// Mitsubishi GX Works2 project: guide_kommunikasjon_master   PLC: Q00

// global labels: Global1
VAR_GLOBAL
  tank AT D0 : INT;
  slider AT D20 : INT;
  knapp_0 AT M20 : BOOL;
  knapp_1 AT M21 : BOOL;
  lampe_0 AT M100 : BOOL;
  lampe_1 AT M101 : BOOL;
  avFlagg_0 AT M0 : BOOL;
  avFlagg_1 AT M1 : BOOL;
  paFlagg_0 AT M10 : BOOL;
  paFlagg_1 AT M11 : BOOL;
END_VAR

// task Task_01 (event TRUE, interval 0, priority 31): POU_01

PROGRAM POU_01
(* structured ladder/FBD written out as ST: instructions are called as NAME(EN, inputs, outputs); _pN, _eN, _tN stand for wires *)
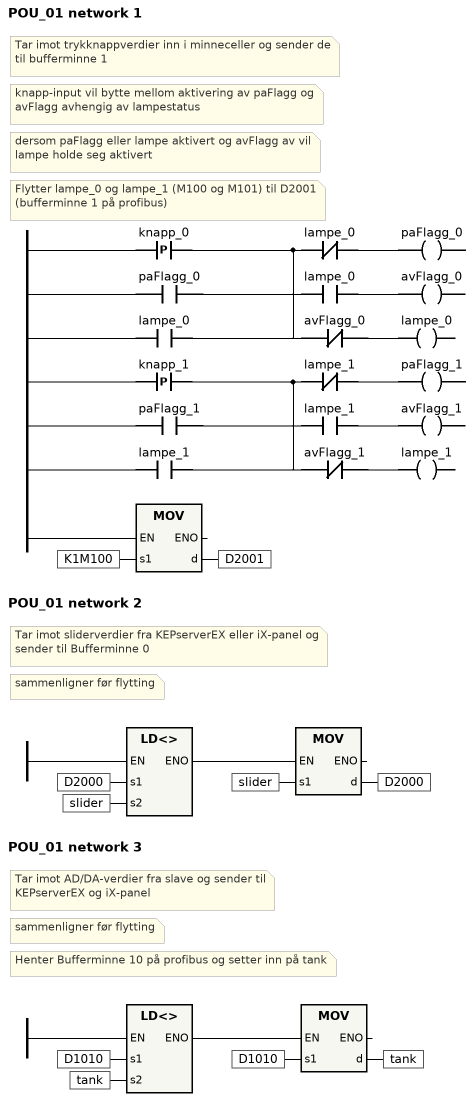
(* network 1 *)
(* Tar imot trykknappverdier inn i minneceller og sender de til bufferminne 1 *)
(* knapp-input vil bytte mellom aktivering av paFlagg og avFlagg avhengig av lampestatus *)
(* dersom paFlagg eller lampe aktivert og avFlagg av vil lampe holde seg aktivert *)
(* Flytter lampe_0 og lampe_1 (M100 og M101) til D2001 (bufferminne 1 på profibus) *)
_p1 := LDP(TRUE, knapp_0);
paFlagg_0 := _p1 AND NOT lampe_0;
avFlagg_0 := _p1 AND lampe_0;
lampe_0 := (paFlagg_0 OR lampe_0) AND NOT avFlagg_0;
_p2 := LDP(TRUE, knapp_1);
paFlagg_1 := _p2 AND NOT lampe_1;
avFlagg_1 := _p2 AND lampe_1;
lampe_1 := (paFlagg_1 OR lampe_1) AND NOT avFlagg_1;
MOV(TRUE, K1M100, D2001);
(* network 2 *)
(* Tar imot sliderverdier fra KEPserverEX eller iX-panel og sender til Bufferminne 0 *)
(* sammenligner før flytting *)
_e1 := LD<>(TRUE, D2000, slider);
MOV(_e1, slider, D2000);
(* network 3 *)
(* Tar imot AD/DA-verdier fra slave og sender til KEPserverEX og iX-panel *)
(* sammenligner før flytting *)
(* Henter Bufferminne 10 på profibus og setter inn på tank *)
_e1 := LD<>(TRUE, D1010, tank);
MOV(_e1, D1010, tank);
END_PROGRAM
